Yaskawa INFORM job: Hexagon_ROBODK.jbi

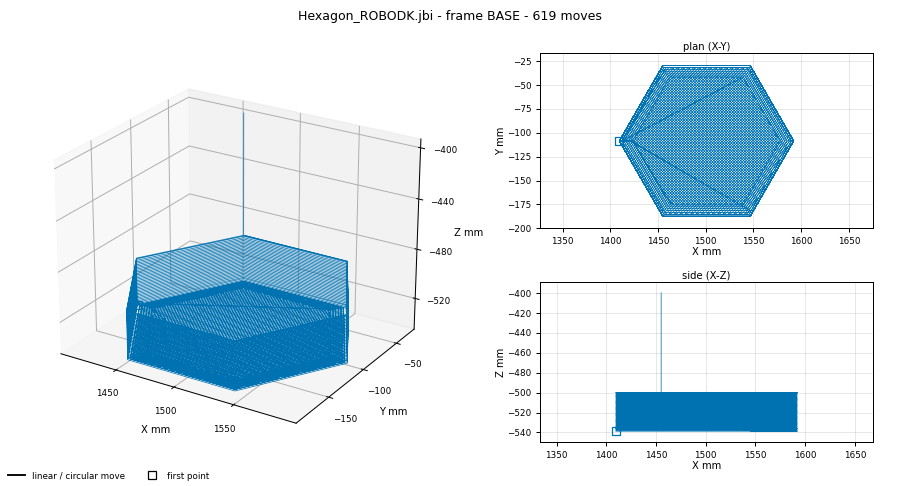
[picture p0: tool path of Hexagon_ROBODK.jbi in frame BASE, 619 of 620 moves have a stored position in this frame; points joined in program order, loops and branches not executed]
/JOB
//NAME HEXAGON
//POS
///NPOS 620,0,0,0,0,0
///TOOL 9
///POSTYPE PULSE
///PULSE
C00000=-4,42,-30,0,-18,-176
///TOOL 9
///POSTYPE BASE
///RECTAN
///RCONF 0,0,0,0,0,0,0,0
C00001=1409.577,-108.483,-538.800,180.00,-0.00,180.00
C00002=1455.188,-29.484,-538.800,180.00,-0.00,-180.00
C00003=1546.406,-29.484,-538.800,180.00,-0.00,-180.00
C00004=1592.017,-108.483,-538.800,180.00,-0.00,180.00
C00005=1546.406,-187.483,-538.800,180.00,0.00,-180.00
C00006=1455.188,-187.483,-538.800,180.00,0.00,-180.00
C00007=1409.577,-108.483,-538.800,180.00,-0.00,180.00
C00008=1410.014,-107.726,-538.800,180.00,0.00,-180.00
C00009=1412.706,-108.484,-538.800,180.00,-0.00,-180.00
C00010=1411.773,-108.482,-538.800,180.00,-0.00,-180.00
C00011=1456.286,-31.385,-538.800,180.00,0.00,-180.00
C00012=1545.308,-31.385,-538.800,180.00,-0.00,-180.00
C00013=1589.821,-108.483,-538.800,180.00,0.00,180.00
C00014=1545.308,-185.582,-538.800,180.00,-0.00,-180.00
C00015=1456.286,-185.582,-538.800,180.00,-0.00,180.00
C00016=1411.773,-108.482,-538.800,180.00,-0.00,-180.00
C00017=1412.706,-108.484,-538.800,180.00,-0.00,-180.00
C00018=1458.101,-32.386,-538.800,180.00,0.00,-180.00
C00019=1455.169,-35.318,-538.800,180.00,0.00,-180.00
C00020=1454.816,-35.671,-538.800,180.00,0.00,180.00
C00021=1460.929,-32.386,-538.800,180.00,0.00,-180.00
C00022=1451.306,-42.010,-538.800,180.00,-0.00,-180.00
C00023=1450.953,-42.363,-538.800,180.00,-0.00,-180.00
C00024=1447.442,-48.702,-538.800,180.00,-0.00,-180.00
C00025=1463.758,-32.386,-538.800,180.00,0.00,180.00
C00026=1466.586,-32.386,-538.800,180.00,0.00,180.00
C00027=1443.578,-55.394,-538.800,180.00,0.00,-180.00
C00028=1443.225,-55.747,-538.800,180.00,0.00,-180.00
C00029=1439.715,-62.086,-538.800,180.00,-0.00,180.00
C00030=1469.415,-32.386,-538.800,180.00,-0.00,-180.00
C00031=1472.243,-32.386,-538.800,180.00,-0.00,-180.00
C00032=1435.850,-68.779,-538.800,180.00,-0.00,-180.00
C00033=1435.497,-69.132,-538.800,180.00,0.00,-180.00
C00034=1431.987,-75.471,-538.800,180.00,0.00,180.00
C00035=1475.071,-32.386,-538.800,180.00,-0.00,-180.00
C00036=1477.900,-32.386,-538.800,180.00,0.00,180.00
C00037=1428.123,-82.163,-538.800,180.00,0.00,180.00
C00038=1427.770,-82.516,-538.800,180.00,0.00,-180.00
C00039=1424.259,-88.855,-538.800,180.00,-0.00,180.00
C00040=1480.728,-32.386,-538.800,180.00,0.00,180.00
C00041=1483.557,-32.386,-538.800,180.00,-0.00,-180.00
C00042=1420.396,-95.547,-538.800,180.00,0.00,180.00
C00043=1420.043,-95.900,-538.800,180.00,-0.00,-180.00
C00044=1416.532,-102.239,-538.800,180.00,0.00,-180.00
C00045=1486.385,-32.386,-538.800,180.00,-0.00,180.00
C00046=1489.214,-32.386,-538.800,180.00,-0.00,180.00
C00047=1412.997,-108.603,-538.800,180.00,0.00,-180.00
C00048=1414.032,-110.396,-538.800,180.00,0.00,-180.00
C00049=1492.042,-32.386,-538.800,180.00,0.00,-180.00
C00050=1494.870,-32.386,-538.800,180.00,0.00,-180.00
C00051=1415.067,-112.190,-538.800,180.00,0.00,-180.00
C00052=1416.102,-113.983,-538.800,180.00,0.00,-180.00
C00053=1497.699,-32.386,-538.800,180.00,0.00,-180.00
C00054=1500.527,-32.386,-538.800,180.00,-0.00,-180.00
C00055=1417.137,-115.776,-538.800,180.00,-0.00,-180.00
C00056=1418.173,-117.569,-538.800,180.00,0.00,180.00
C00057=1503.356,-32.386,-538.800,180.00,0.00,-180.00
C00058=1506.184,-32.386,-538.800,180.00,-0.00,-180.00
C00059=1419.208,-119.362,-538.800,180.00,0.00,-180.00
C00060=1420.243,-121.156,-538.800,180.00,-0.00,-180.00
C00061=1509.013,-32.386,-538.800,180.00,-0.00,-180.00
C00062=1511.841,-32.386,-538.800,180.00,0.00,180.00
C00063=1421.278,-122.949,-538.800,180.00,0.00,-180.00
C00064=1422.313,-124.742,-538.800,180.00,-0.00,-180.00
C00065=1514.669,-32.386,-538.800,180.00,-0.00,-180.00
C00066=1517.498,-32.386,-538.800,180.00,0.00,-180.00
C00067=1423.349,-126.535,-538.800,180.00,-0.00,-180.00
C00068=1424.384,-128.329,-538.800,180.00,0.00,180.00
C00069=1520.326,-32.386,-538.800,180.00,-0.00,-180.00
C00070=1523.155,-32.386,-538.800,180.00,0.00,-180.00
C00071=1425.419,-130.122,-538.800,180.00,-0.00,180.00
C00072=1426.455,-131.914,-538.800,180.00,-0.00,-180.00
C00073=1525.983,-32.386,-538.800,180.00,0.00,-180.00
C00074=1528.812,-32.386,-538.800,180.00,-0.00,-180.00
C00075=1427.490,-133.708,-538.800,180.00,0.00,-180.00
C00076=1428.525,-135.501,-538.800,180.00,0.00,-180.00
C00077=1531.640,-32.386,-538.800,180.00,-0.00,180.00
C00078=1534.468,-32.386,-538.800,180.00,0.00,-180.00
C00079=1429.561,-137.294,-538.800,180.00,0.00,-180.00
C00080=1430.596,-139.087,-538.800,180.00,-0.00,180.00
C00081=1537.297,-32.386,-538.800,180.00,-0.00,-180.00
C00082=1540.125,-32.386,-538.800,180.00,0.00,-180.00
C00083=1431.631,-140.880,-538.800,180.00,0.00,180.00
C00084=1432.666,-142.674,-538.800,180.00,0.00,180.00
C00085=1542.954,-32.386,-538.800,180.00,-0.00,-180.00
C00086=1545.115,-33.053,-538.800,180.00,-0.00,-180.00
C00087=1433.701,-144.467,-538.800,180.00,-0.00,-180.00
C00088=1434.737,-146.260,-538.800,180.00,-0.00,-180.00
C00089=1546.150,-34.846,-538.800,180.00,0.00,-180.00
C00090=1547.186,-36.639,-538.800,180.00,0.00,180.00
C00091=1435.772,-148.053,-538.800,180.00,-0.00,-180.00
C00092=1436.807,-149.847,-538.800,180.00,0.00,-180.00
C00093=1548.221,-38.433,-538.800,180.00,-0.00,-180.00
C00094=1549.257,-40.225,-538.800,180.00,0.00,-180.00
C00095=1437.842,-151.640,-538.800,180.00,0.00,180.00
C00096=1438.877,-153.433,-538.800,180.00,-0.00,-180.00
C00097=1550.292,-42.018,-538.800,180.00,0.00,180.00
C00098=1551.327,-43.812,-538.800,180.00,0.00,-180.00
C00099=1439.913,-155.226,-538.800,180.00,0.00,-180.00
C00100=1440.949,-157.019,-538.800,180.00,0.00,180.00
C00101=1552.362,-45.605,-538.800,180.00,0.00,180.00
C00102=1553.398,-47.398,-538.800,180.00,-0.00,-180.00
C00103=1441.984,-158.812,-538.800,180.00,-0.00,-180.00
C00104=1443.019,-160.605,-538.800,180.00,0.00,-180.00
C00105=1554.433,-49.191,-538.800,180.00,0.00,-180.00
C00106=1555.468,-50.985,-538.800,180.00,0.00,-180.00
C00107=1444.054,-162.398,-538.800,180.00,-0.00,-180.00
C00108=1445.089,-164.192,-538.800,180.00,-0.00,180.00
C00109=1556.503,-52.778,-538.800,180.00,-0.00,180.00
C00110=1557.538,-54.571,-538.800,180.00,-0.00,-180.00
C00111=1446.125,-165.985,-538.800,180.00,0.00,-180.00
C00112=1447.160,-167.778,-538.800,180.00,0.00,-180.00
C00113=1558.574,-56.364,-538.800,180.00,0.00,-180.00
C00114=1559.610,-58.157,-538.800,180.00,-0.00,180.00
C00115=1448.195,-169.571,-538.800,180.00,-0.00,-180.00
C00116=1449.230,-171.365,-538.800,180.00,0.00,180.00
C00117=1560.645,-59.950,-538.800,180.00,0.00,-180.00
C00118=1561.680,-61.743,-538.800,180.00,0.00,-180.00
C00119=1450.265,-173.158,-538.800,180.00,0.00,180.00
C00120=1451.301,-174.951,-538.800,180.00,-0.00,-180.00
C00121=1562.715,-63.536,-538.800,180.00,0.00,180.00
C00122=1563.750,-65.330,-538.800,180.00,0.00,-180.00
C00123=1452.336,-176.744,-538.800,180.00,-0.00,-180.00
C00124=1453.371,-178.537,-538.800,180.00,-0.00,-180.00
C00125=1564.786,-67.123,-538.800,180.00,0.00,-180.00
C00126=1565.821,-68.916,-538.800,180.00,-0.00,-180.00
C00127=1454.406,-180.331,-538.800,180.00,0.00,-180.00
C00128=1455.442,-182.123,-538.800,180.00,-0.00,-180.00
C00129=1566.857,-70.709,-538.800,180.00,0.00,180.00
C00130=1567.892,-72.502,-538.800,180.00,-0.00,-180.00
C00131=1456.477,-183.916,-538.800,180.00,0.00,-180.00
C00132=1458.640,-184.582,-538.800,180.00,0.00,180.00
C00133=1568.927,-74.295,-538.800,180.00,0.00,-180.00
C00134=1569.962,-76.088,-538.800,180.00,0.00,-180.00
C00135=1461.468,-184.582,-538.800,180.00,-0.00,-180.00
C00136=1464.297,-184.582,-538.800,180.00,0.00,-180.00
C00137=1570.998,-77.881,-538.800,180.00,-0.00,180.00
C00138=1572.033,-79.675,-538.800,180.00,0.00,-180.00
C00139=1467.125,-184.582,-538.800,180.00,-0.00,-180.00
C00140=1469.953,-184.582,-538.800,180.00,0.00,180.00
C00141=1573.068,-81.468,-538.800,180.00,-0.00,-180.00
C00142=1574.103,-83.261,-538.800,180.00,-0.00,-180.00
C00143=1472.782,-184.582,-538.800,180.00,-0.00,180.00
C00144=1475.610,-184.582,-538.800,180.00,0.00,-180.00
C00145=1575.138,-85.054,-538.800,180.00,0.00,180.00
C00146=1576.174,-86.847,-538.800,180.00,0.00,-180.00
C00147=1478.439,-184.582,-538.800,180.00,0.00,-180.00
C00148=1481.267,-184.582,-538.800,180.00,0.00,-180.00
C00149=1577.209,-88.640,-538.800,180.00,-0.00,-180.00
C00150=1578.245,-90.433,-538.800,180.00,-0.00,-180.00
C00151=1484.095,-184.582,-538.800,180.00,0.00,-180.00
C00152=1486.924,-184.582,-538.800,180.00,-0.00,180.00
C00153=1579.280,-92.227,-538.800,180.00,0.00,-180.00
C00154=1580.315,-94.020,-538.800,180.00,0.00,-180.00
C00155=1489.752,-184.582,-538.800,180.00,0.00,-180.00
C00156=1492.581,-184.582,-538.800,180.00,-0.00,-180.00
C00157=1581.350,-95.813,-538.800,180.00,-0.00,-180.00
C00158=1582.385,-97.606,-538.800,180.00,0.00,180.00
C00159=1495.409,-184.582,-538.800,180.00,-0.00,-180.00
C00160=1498.238,-184.582,-538.800,180.00,0.00,180.00
C00161=1583.421,-99.399,-538.800,180.00,0.00,-180.00
C00162=1584.456,-101.193,-538.800,180.00,-0.00,-180.00
C00163=1501.066,-184.582,-538.800,180.00,0.00,-180.00
C00164=1503.894,-184.582,-538.800,180.00,-0.00,-180.00
C00165=1585.492,-102.985,-538.800,180.00,0.00,180.00
C00166=1586.527,-104.778,-538.800,180.00,0.00,-180.00
C00167=1506.723,-184.582,-538.800,180.00,-0.00,-180.00
C00168=1509.551,-184.582,-538.800,180.00,0.00,-180.00
C00169=1587.562,-106.572,-538.800,180.00,0.00,-180.00
C00170=1588.597,-108.365,-538.800,180.00,0.00,-180.00
C00171=1512.380,-184.582,-538.800,180.00,0.00,-180.00
C00172=1515.208,-184.582,-538.800,180.00,0.00,-180.00
C00173=1585.057,-114.734,-538.800,180.00,0.00,180.00
C00174=1585.410,-114.381,-538.800,180.00,0.00,-180.00
C00175=1581.193,-121.426,-538.800,180.00,-0.00,-180.00
C00176=1518.037,-184.582,-538.800,180.00,-0.00,-180.00
C00177=1520.865,-184.582,-538.800,180.00,-0.00,-180.00
C00178=1577.330,-128.118,-538.800,180.00,0.00,-180.00
C00179=1577.683,-127.765,-538.800,180.00,0.00,-180.00
C00180=1573.466,-134.810,-538.800,180.00,-0.00,-180.00
C00181=1523.693,-184.582,-538.800,180.00,-0.00,-180.00
C00182=1526.522,-184.582,-538.800,180.00,0.00,-180.00
C00183=1569.602,-141.502,-538.800,180.00,0.00,180.00
C00184=1569.955,-141.149,-538.800,180.00,0.00,180.00
C00185=1565.739,-148.194,-538.800,180.00,0.00,-180.00
C00186=1529.350,-184.582,-538.800,180.00,0.00,-180.00
C00187=1532.179,-184.582,-538.800,180.00,0.00,-180.00
C00188=1561.875,-154.886,-538.800,180.00,-0.00,-180.00
C00189=1562.228,-154.533,-538.800,180.00,0.00,180.00
C00190=1558.011,-161.578,-538.800,180.00,0.00,-180.00
C00191=1535.007,-184.582,-538.800,180.00,0.00,-180.00
C00192=1537.836,-184.582,-538.800,180.00,-0.00,180.00
C00193=1554.148,-168.270,-538.800,180.00,-0.00,-180.00
C00194=1554.501,-167.917,-538.800,180.00,-0.00,-180.00
C00195=1550.284,-174.962,-538.800,180.00,-0.00,-180.00
C00196=1540.664,-184.582,-538.800,180.00,-0.00,-180.00
C00197=1543.492,-184.582,-538.800,180.00,0.00,-180.00
C00198=1546.421,-181.654,-538.800,180.00,0.00,-180.00
C00199=1546.774,-181.301,-538.800,180.00,-0.00,180.00
C00200=1545.171,-180.377,-538.800,180.00,-0.00,-180.00
C00201=1545.171,-180.377,-537.600,180.00,0.00,-180.00
C00202=1421.124,-108.483,-537.600,180.00,0.00,180.00
C00203=1441.043,-73.984,-537.600,180.00,0.00,-180.00
C00204=1460.961,-39.484,-537.600,180.00,0.00,180.00
C00205=1540.633,-39.484,-537.600,180.00,0.00,-180.00
C00206=1580.470,-108.483,-537.600,180.00,0.00,-180.00
C00207=1540.633,-177.483,-537.600,180.00,-0.00,-180.00
C00208=1460.961,-177.483,-537.600,180.00,0.00,180.00
C00209=1421.124,-108.483,-537.600,180.00,0.00,180.00
C00210=1418.815,-108.483,-537.600,180.00,0.00,-180.00
C00211=1439.311,-72.984,-537.600,180.00,-0.00,-180.00
C00212=1459.807,-37.484,-537.600,180.00,0.00,-180.00
C00213=1541.787,-37.484,-537.600,180.00,0.00,-180.00
C00214=1582.779,-108.483,-537.600,180.00,0.00,180.00
C00215=1541.787,-179.483,-537.600,180.00,0.00,180.00
C00216=1459.807,-179.483,-537.600,180.00,0.00,-180.00
C00217=1418.815,-108.483,-537.600,180.00,0.00,-180.00
C00218=1416.506,-108.483,-537.600,180.00,-0.00,-180.00
C00219=1437.579,-71.984,-537.600,180.00,-0.00,-180.00
C00220=1458.652,-35.484,-537.600,180.00,0.00,180.00
C00221=1542.942,-35.484,-537.600,180.00,0.00,180.00
C00222=1585.088,-108.483,-537.600,180.00,-0.00,-180.00
C00223=1542.942,-181.483,-537.600,180.00,-0.00,-180.00
C00224=1458.652,-181.483,-537.600,180.00,0.00,-180.00
C00225=1416.506,-108.483,-537.600,180.00,-0.00,-180.00
C00226=1414.196,-108.483,-537.600,180.00,-0.00,180.00
C00227=1435.847,-70.984,-537.600,180.00,-0.00,-180.00
C00228=1457.497,-33.484,-537.600,180.00,0.00,-180.00
C00229=1544.097,-33.484,-537.600,180.00,0.00,-180.00
C00230=1587.398,-108.483,-537.600,180.00,0.00,180.00
C00231=1544.097,-183.483,-537.600,180.00,0.00,-180.00
C00232=1457.497,-183.483,-537.600,180.00,-0.00,-180.00
C00233=1414.196,-108.483,-537.600,180.00,-0.00,180.00
C00234=1412.706,-108.484,-537.600,180.00,0.00,-180.00
C00235=1411.887,-108.483,-537.600,180.00,-0.00,-180.00
C00236=1434.115,-69.984,-537.600,180.00,-0.00,180.00
C00237=1456.343,-31.484,-537.600,180.00,0.00,-180.00
C00238=1545.251,-31.484,-537.600,180.00,0.00,-180.00
C00239=1589.707,-108.483,-537.600,180.00,0.00,-180.00
C00240=1545.251,-185.483,-537.600,180.00,0.00,180.00
C00241=1456.343,-185.483,-537.600,180.00,0.00,-180.00
C00242=1411.887,-108.483,-537.600,180.00,-0.00,-180.00
C00243=1412.706,-108.484,-537.600,180.00,0.00,-180.00
C00244=1409.577,-108.483,-537.600,180.00,0.00,180.00
C00245=1432.383,-68.984,-537.600,180.00,-0.00,-180.00
C00246=1455.188,-29.484,-537.600,180.00,0.00,-180.00
C00247=1546.406,-29.484,-537.600,180.00,0.00,-180.00
C00248=1592.017,-108.483,-537.600,180.00,0.00,180.00
C00249=1546.406,-187.483,-537.600,180.00,0.00,-180.00
C00250=1455.188,-187.483,-537.600,180.00,0.00,-180.00
C00251=1409.577,-108.483,-537.600,180.00,0.00,180.00
C00252=1410.014,-107.726,-537.600,180.00,0.00,-180.00
C00253=1412.706,-108.484,-537.600,180.00,0.00,-180.00
C00254=1423.320,-108.483,-537.600,180.00,-0.00,180.00
C00255=1462.060,-41.384,-537.600,180.00,0.00,-180.00
C00256=1539.534,-41.384,-537.600,180.00,-0.00,-180.00
C00257=1578.274,-108.482,-537.600,180.00,0.00,180.00
C00258=1539.534,-175.582,-537.600,180.00,-0.00,-180.00
C00259=1462.060,-175.582,-537.600,180.00,0.00,-180.00
C00260=1423.320,-108.483,-537.600,180.00,-0.00,180.00
C00261=1463.506,-174.583,-537.600,180.00,0.00,-180.00
C00262=1461.448,-172.525,-537.600,180.00,0.00,-180.00
C00263=1466.334,-174.583,-537.600,180.00,-0.00,-180.00
C00264=1457.585,-165.833,-537.600,180.00,0.00,180.00
C00265=1457.232,-165.480,-537.600,180.00,0.00,-180.00
C00266=1453.721,-159.141,-537.600,180.00,-0.00,-180.00
C00267=1469.163,-174.583,-537.600,180.00,-0.00,-180.00
C00268=1471.991,-174.583,-537.600,180.00,0.00,180.00
C00269=1449.857,-152.449,-537.600,180.00,0.00,-180.00
C00270=1449.504,-152.096,-537.600,180.00,0.00,-180.00
C00271=1445.994,-145.757,-537.600,180.00,-0.00,-180.00
C00272=1474.820,-174.583,-537.600,180.00,0.00,180.00
C00273=1477.648,-174.583,-537.600,180.00,0.00,-180.00
C00274=1442.130,-139.065,-537.600,180.00,-0.00,-180.00
C00275=1441.777,-138.712,-537.600,180.00,-0.00,180.00
C00276=1438.266,-132.373,-537.600,180.00,0.00,-180.00
C00277=1480.477,-174.583,-537.600,180.00,0.00,-180.00
C00278=1483.305,-174.583,-537.600,180.00,-0.00,180.00
C00279=1434.403,-125.680,-537.600,180.00,-0.00,-180.00
C00280=1434.050,-125.327,-537.600,180.00,0.00,180.00
C00281=1430.539,-118.988,-537.600,180.00,0.00,180.00
C00282=1486.133,-174.583,-537.600,180.00,0.00,180.00
C00283=1488.962,-174.583,-537.600,180.00,-0.00,-180.00
C00284=1426.675,-112.296,-537.600,180.00,-0.00,-180.00
C00285=1426.322,-111.943,-537.600,180.00,0.00,-180.00
C00286=1424.921,-107.713,-537.600,180.00,0.00,-180.00
C00287=1491.790,-174.583,-537.600,180.00,0.00,-180.00
C00288=1494.619,-174.583,-537.600,180.00,0.00,-180.00
C00289=1425.956,-105.920,-537.600,180.00,-0.00,-180.00
C00290=1426.991,-104.126,-537.600,180.00,-0.00,-180.00
C00291=1497.447,-174.583,-537.600,180.00,-0.00,-180.00
C00292=1500.276,-174.583,-537.600,180.00,-0.00,-180.00
C00293=1428.026,-102.333,-537.600,180.00,-0.00,-180.00
C00294=1429.061,-100.540,-537.600,180.00,-0.00,180.00
C00295=1503.104,-174.583,-537.600,180.00,-0.00,-180.00
C00296=1505.932,-174.583,-537.600,180.00,-0.00,180.00
C00297=1430.097,-98.747,-537.600,180.00,0.00,-180.00
C00298=1431.132,-96.954,-537.600,180.00,-0.00,180.00
C00299=1508.761,-174.583,-537.600,180.00,0.00,-180.00
C00300=1511.589,-174.583,-537.600,180.00,-0.00,-180.00
C00301=1432.168,-95.161,-537.600,180.00,0.00,180.00
C00302=1433.203,-93.368,-537.600,180.00,-0.00,-180.00
C00303=1514.418,-174.583,-537.600,180.00,-0.00,180.00
C00304=1517.246,-174.583,-537.600,180.00,0.00,-180.00
C00305=1434.238,-91.575,-537.600,180.00,0.00,180.00
C00306=1435.273,-89.781,-537.600,180.00,-0.00,-180.00
C00307=1520.075,-174.583,-537.600,180.00,-0.00,-180.00
C00308=1522.903,-174.583,-537.600,180.00,-0.00,-180.00
C00309=1436.309,-87.988,-537.600,180.00,-0.00,-180.00
C00310=1437.344,-86.195,-537.600,180.00,-0.00,-180.00
C00311=1525.731,-174.583,-537.600,180.00,0.00,180.00
C00312=1528.560,-174.583,-537.600,180.00,-0.00,180.00
C00313=1438.379,-84.402,-537.600,180.00,-0.00,-180.00
C00314=1439.414,-82.608,-537.600,180.00,0.00,180.00
C00315=1531.388,-174.583,-537.600,180.00,0.00,-180.00
C00316=1534.217,-174.583,-537.600,180.00,-0.00,-180.00
C00317=1440.449,-80.815,-537.600,180.00,0.00,180.00
C00318=1441.485,-79.023,-537.600,180.00,0.00,-180.00
C00319=1537.045,-174.583,-537.600,180.00,0.00,-180.00
C00320=1539.292,-174.001,-537.600,180.00,-0.00,180.00
C00321=1442.520,-77.230,-537.600,180.00,0.00,-180.00
C00322=1443.556,-75.436,-537.600,180.00,-0.00,-180.00
C00323=1540.327,-172.207,-537.600,180.00,-0.00,-180.00
C00324=1541.362,-170.414,-537.600,180.00,0.00,180.00
C00325=1444.591,-73.643,-537.600,180.00,0.00,-180.00
C00326=1445.626,-71.850,-537.600,180.00,0.00,-180.00
C00327=1542.397,-168.621,-537.600,180.00,0.00,-180.00
C00328=1543.432,-166.828,-537.600,180.00,0.00,-180.00
C00329=1446.661,-70.057,-537.600,180.00,-0.00,180.00
C00330=1447.696,-68.263,-537.600,180.00,0.00,180.00
C00331=1544.468,-165.035,-537.600,180.00,0.00,180.00
C00332=1545.503,-163.241,-537.600,180.00,0.00,-180.00
C00333=1448.732,-66.470,-537.600,180.00,-0.00,-180.00
C00334=1449.767,-64.677,-537.600,180.00,0.00,180.00
C00335=1546.538,-161.448,-537.600,180.00,-0.00,-180.00
C00336=1547.573,-159.655,-537.600,180.00,-0.00,-180.00
C00337=1450.803,-62.884,-537.600,180.00,-0.00,-180.00
C00338=1451.838,-61.091,-537.600,180.00,0.00,180.00
C00339=1548.608,-157.862,-537.600,180.00,-0.00,-180.00
C00340=1549.644,-156.068,-537.600,180.00,-0.00,-180.00
C00341=1452.873,-59.298,-537.600,180.00,-0.00,180.00
C00342=1453.908,-57.505,-537.600,180.00,0.00,180.00
C00343=1550.679,-154.275,-537.600,180.00,-0.00,-180.00
C00344=1551.715,-152.483,-537.600,180.00,0.00,-180.00
C00345=1454.944,-55.712,-537.600,180.00,-0.00,-180.00
C00346=1455.979,-53.918,-537.600,180.00,0.00,-180.00
C00347=1552.750,-150.689,-537.600,180.00,0.00,-180.00
C00348=1553.785,-148.896,-537.600,180.00,-0.00,-180.00
C00349=1457.014,-52.125,-537.600,180.00,0.00,-180.00
C00350=1458.049,-50.332,-537.600,180.00,-0.00,-180.00
C00351=1554.820,-147.103,-537.600,180.00,-0.00,-180.00
C00352=1555.856,-145.310,-537.600,180.00,0.00,-180.00
C00353=1459.084,-48.539,-537.600,180.00,0.00,-180.00
C00354=1460.120,-46.746,-537.600,180.00,-0.00,-180.00
C00355=1556.891,-143.517,-537.600,180.00,0.00,180.00
C00356=1557.926,-141.723,-537.600,180.00,0.00,-180.00
C00357=1461.156,-44.953,-537.600,180.00,-0.00,-180.00
C00358=1462.191,-43.160,-537.600,180.00,-0.00,-180.00
C00359=1558.961,-139.930,-537.600,180.00,0.00,180.00
C00360=1559.996,-138.137,-537.600,180.00,-0.00,180.00
C00361=1464.245,-42.385,-537.600,180.00,0.00,180.00
C00362=1467.073,-42.385,-537.600,180.00,0.00,-180.00
C00363=1561.032,-136.344,-537.600,180.00,-0.00,-180.00
C00364=1562.067,-134.550,-537.600,180.00,-0.00,-180.00
C00365=1469.902,-42.385,-537.600,180.00,-0.00,-180.00
C00366=1472.730,-42.385,-537.600,180.00,0.00,-180.00
C00367=1563.102,-132.757,-537.600,180.00,-0.00,180.00
C00368=1564.138,-130.965,-537.600,180.00,-0.00,180.00
C00369=1475.559,-42.385,-537.600,180.00,0.00,-180.00
C00370=1478.387,-42.385,-537.600,180.00,0.00,-180.00
C00371=1565.173,-129.171,-537.600,180.00,-0.00,180.00
C00372=1566.208,-127.378,-537.600,180.00,0.00,-180.00
C00373=1481.215,-42.385,-537.600,180.00,0.00,-180.00
C00374=1484.044,-42.385,-537.600,180.00,0.00,-180.00
C00375=1567.243,-125.585,-537.600,180.00,0.00,180.00
C00376=1568.279,-123.792,-537.600,180.00,0.00,-180.00
C00377=1486.872,-42.385,-537.600,180.00,0.00,-180.00
C00378=1489.701,-42.385,-537.600,180.00,0.00,180.00
C00379=1569.314,-121.999,-537.600,180.00,0.00,-180.00
C00380=1570.349,-120.205,-537.600,180.00,0.00,-180.00
C00381=1492.529,-42.385,-537.600,180.00,0.00,-180.00
C00382=1495.358,-42.385,-537.600,180.00,0.00,-180.00
C00383=1571.384,-118.412,-537.600,180.00,-0.00,-180.00
C00384=1572.420,-116.619,-537.600,180.00,0.00,180.00
C00385=1498.186,-42.385,-537.600,180.00,0.00,-180.00
C00386=1501.014,-42.385,-537.600,180.00,0.00,-180.00
C00387=1573.455,-114.826,-537.600,180.00,-0.00,-180.00
C00388=1574.490,-113.032,-537.600,180.00,0.00,180.00
C00389=1503.843,-42.385,-537.600,180.00,-0.00,-180.00
C00390=1506.671,-42.385,-537.600,180.00,0.00,-180.00
C00391=1575.525,-111.239,-537.600,180.00,0.00,-180.00
C00392=1576.561,-109.447,-537.600,180.00,0.00,180.00
C00393=1509.500,-42.385,-537.600,180.00,0.00,-180.00
C00394=1512.328,-42.385,-537.600,180.00,-0.00,-180.00
C00395=1575.330,-105.387,-537.600,180.00,-0.00,-180.00
C00396=1575.683,-105.740,-537.600,180.00,0.00,-180.00
C00397=1571.466,-98.695,-537.600,180.00,0.00,-180.00
C00398=1515.157,-42.385,-537.600,180.00,0.00,-180.00
C00399=1517.985,-42.385,-537.600,180.00,-0.00,-180.00
C00400=1567.603,-92.003,-537.600,180.00,0.00,-180.00
C00401=1567.956,-92.356,-537.600,180.00,0.00,-180.00
C00402=1563.739,-85.311,-537.600,180.00,0.00,-180.00
C00403=1520.813,-42.385,-537.600,180.00,-0.00,-180.00
C00404=1523.642,-42.385,-537.600,180.00,-0.00,180.00
C00405=1559.875,-78.619,-537.600,180.00,-0.00,180.00
C00406=1560.228,-78.972,-537.600,180.00,-0.00,180.00
C00407=1556.012,-71.927,-537.600,180.00,0.00,180.00
C00408=1526.470,-42.385,-537.600,180.00,0.00,-180.00
C00409=1529.299,-42.385,-537.600,180.00,-0.00,180.00
C00410=1552.148,-65.235,-537.600,180.00,0.00,-180.00
C00411=1552.501,-65.588,-537.600,180.00,-0.00,180.00
C00412=1548.285,-58.543,-537.600,180.00,0.00,-180.00
C00413=1532.127,-42.385,-537.600,180.00,-0.00,180.00
C00414=1534.956,-42.385,-537.600,180.00,-0.00,180.00
C00415=1544.421,-51.851,-537.600,180.00,0.00,-180.00
C00416=1544.774,-52.204,-537.600,180.00,0.00,180.00
C00417=1540.557,-45.159,-537.600,180.00,0.00,180.00
C00418=1537.784,-42.385,-537.600,180.00,-0.00,180.00
C00419=1537.784,-42.385,-536.400,180.00,0.00,180.00
C00420=1412.706,-108.484,-536.400,180.00,-0.00,-180.00
C00421=1409.576,-108.484,-536.400,180.00,-0.00,-180.00
C00422=1455.186,-187.484,-536.400,180.00,-0.00,-180.00
C00423=1546.408,-187.484,-536.400,180.00,0.00,180.00
C00424=1592.018,-108.484,-536.400,180.00,0.00,180.00
C00425=1546.408,-29.484,-536.400,180.00,0.00,-180.00
C00426=1455.186,-29.484,-536.400,180.00,-0.00,-180.00
C00427=1409.576,-108.484,-536.400,180.00,-0.00,-180.00
C00428=1455.186,-187.484,-536.200,180.00,0.00,-180.00
C00429=1546.408,-187.484,-536.000,180.00,0.00,180.00
C00430=1592.018,-108.484,-535.800,180.00,-0.00,180.00
C00431=1546.408,-29.484,-535.600,180.00,0.00,-180.00
C00432=1455.186,-29.484,-535.400,180.00,-0.00,-180.00
C00433=1409.576,-108.484,-535.200,180.00,-0.00,-180.00
C00434=1455.186,-187.484,-535.000,180.00,0.00,-180.00
C00435=1546.408,-187.484,-534.800,180.00,-0.00,-180.00
C00436=1592.018,-108.484,-534.600,180.00,-0.00,180.00
C00437=1546.408,-29.484,-534.400,180.00,-0.00,-180.00
C00438=1455.186,-29.484,-534.200,180.00,0.00,-180.00
C00439=1409.576,-108.484,-534.000,180.00,0.00,-180.00
C00440=1455.186,-187.484,-533.800,180.00,0.00,-180.00
C00441=1546.408,-187.484,-533.600,180.00,0.00,-180.00
C00442=1592.018,-108.484,-533.400,180.00,0.00,180.00
C00443=1546.408,-29.484,-533.200,180.00,-0.00,-180.00
C00444=1455.186,-29.484,-533.000,180.00,-0.00,-180.00
C00445=1409.576,-108.484,-532.800,180.00,0.00,-180.00
C00446=1455.186,-187.484,-532.600,180.00,0.00,-180.00
C00447=1546.408,-187.484,-532.400,180.00,0.00,-180.00
C00448=1592.018,-108.484,-532.200,180.00,-0.00,180.00
C00449=1546.408,-29.484,-532.000,180.00,0.00,-180.00
C00450=1455.186,-29.484,-531.800,180.00,0.00,-180.00
C00451=1409.576,-108.484,-531.600,180.00,-0.00,-180.00
C00452=1455.186,-187.484,-531.400,180.00,-0.00,-180.00
C00453=1546.408,-187.484,-531.200,180.00,0.00,-180.00
C00454=1592.018,-108.484,-531.000,180.00,-0.00,180.00
C00455=1546.408,-29.484,-530.800,180.00,0.00,-180.00
C00456=1455.186,-29.484,-530.600,180.00,0.00,-180.00
C00457=1409.576,-108.484,-530.400,180.00,0.00,-180.00
C00458=1455.186,-187.484,-530.200,180.00,0.00,-180.00
C00459=1546.408,-187.484,-530.000,180.00,0.00,180.00
C00460=1592.018,-108.484,-529.800,180.00,0.00,180.00
C00461=1546.408,-29.484,-529.600,180.00,0.00,-180.00
C00462=1455.186,-29.484,-529.400,180.00,-0.00,-180.00
C00463=1409.576,-108.484,-529.200,180.00,-0.00,-180.00
C00464=1455.186,-187.484,-529.000,180.00,-0.00,-180.00
C00465=1546.408,-187.484,-528.800,180.00,-0.00,180.00
C00466=1592.018,-108.484,-528.600,180.00,0.00,180.00
C00467=1546.408,-29.484,-528.400,180.00,0.00,-180.00
C00468=1455.186,-29.484,-528.200,180.00,0.00,-180.00
C00469=1409.576,-108.484,-528.000,180.00,-0.00,-180.00
C00470=1455.186,-187.484,-527.800,180.00,-0.00,-180.00
C00471=1546.408,-187.484,-527.600,180.00,-0.00,-180.00
C00472=1592.018,-108.484,-527.400,180.00,-0.00,180.00
C00473=1546.408,-29.484,-527.200,180.00,0.00,-180.00
C00474=1455.186,-29.484,-527.000,180.00,0.00,-180.00
C00475=1409.576,-108.484,-526.800,180.00,0.00,-180.00
C00476=1455.186,-187.484,-526.600,180.00,0.00,-180.00
C00477=1546.408,-187.484,-526.400,180.00,-0.00,-180.00
C00478=1592.018,-108.484,-526.200,180.00,-0.00,180.00
C00479=1546.408,-29.484,-526.000,180.00,-0.00,-180.00
C00480=1455.186,-29.484,-525.800,180.00,0.00,-180.00
C00481=1409.576,-108.484,-525.600,180.00,0.00,-180.00
C00482=1455.186,-187.484,-525.400,180.00,0.00,-180.00
C00483=1546.408,-187.484,-525.200,180.00,-0.00,-180.00
C00484=1592.018,-108.484,-525.000,180.00,0.00,180.00
C00485=1546.408,-29.484,-524.800,180.00,-0.00,-180.00
C00486=1455.186,-29.484,-524.600,180.00,-0.00,-180.00
C00487=1409.576,-108.484,-524.400,180.00,0.00,-180.00
C00488=1455.186,-187.484,-524.200,180.00,0.00,-180.00
C00489=1546.408,-187.484,-524.000,180.00,0.00,-180.00
C00490=1592.018,-108.484,-523.800,180.00,-0.00,180.00
C00491=1546.408,-29.484,-523.600,180.00,0.00,-180.00
C00492=1455.186,-29.484,-523.400,180.00,0.00,-180.00
C00493=1409.576,-108.484,-523.200,180.00,-0.00,-180.00
C00494=1455.186,-187.484,-523.000,180.00,-0.00,-180.00
C00495=1546.408,-187.484,-522.800,180.00,0.00,180.00
C00496=1592.018,-108.484,-522.600,180.00,-0.00,180.00
C00497=1546.408,-29.484,-522.400,180.00,-0.00,-180.00
C00498=1455.186,-29.484,-522.200,180.00,0.00,-180.00
C00499=1409.576,-108.484,-522.000,180.00,0.00,-180.00
C00500=1455.186,-187.484,-521.800,180.00,-0.00,-180.00
C00501=1546.408,-187.484,-521.600,180.00,0.00,-180.00
C00502=1592.018,-108.484,-521.400,180.00,0.00,180.00
C00503=1546.408,-29.484,-521.200,180.00,0.00,-180.00
C00504=1455.186,-29.484,-521.000,180.00,0.00,-180.00
C00505=1409.576,-108.484,-520.800,180.00,-0.00,-180.00
C00506=1455.186,-187.484,-520.600,180.00,-0.00,-180.00
C00507=1546.408,-187.484,-520.400,180.00,-0.00,-180.00
C00508=1592.018,-108.484,-520.200,180.00,0.00,180.00
C00509=1546.408,-29.484,-520.000,180.00,-0.00,-180.00
C00510=1455.186,-29.484,-519.800,180.00,-0.00,-180.00
C00511=1409.576,-108.484,-519.600,180.00,0.00,-180.00
C00512=1455.186,-187.484,-519.400,180.00,0.00,-180.00
C00513=1546.408,-187.484,-519.200,180.00,0.00,-180.00
C00514=1592.018,-108.484,-519.000,180.00,-0.00,180.00
C00515=1546.408,-29.484,-518.800,180.00,0.00,-180.00
C00516=1455.186,-29.484,-518.600,180.00,-0.00,-180.00
C00517=1409.576,-108.484,-518.400,180.00,-0.00,-180.00
C00518=1455.186,-187.484,-518.200,180.00,-0.00,-180.00
C00519=1546.408,-187.484,-518.000,180.00,-0.00,-180.00
C00520=1592.018,-108.484,-517.800,180.00,-0.00,180.00
C00521=1546.408,-29.484,-517.600,180.00,-0.00,-180.00
C00522=1455.186,-29.484,-517.400,180.00,-0.00,-180.00
C00523=1409.576,-108.484,-517.200,180.00,-0.00,-180.00
C00524=1455.186,-187.484,-517.000,180.00,0.00,-180.00
C00525=1546.408,-187.484,-516.800,180.00,-0.00,-180.00
C00526=1592.018,-108.484,-516.600,180.00,0.00,180.00
C00527=1546.408,-29.484,-516.400,180.00,0.00,-180.00
C00528=1455.186,-29.484,-516.200,180.00,-0.00,-180.00
C00529=1409.576,-108.484,-516.000,180.00,0.00,-180.00
C00530=1455.186,-187.484,-515.800,180.00,-0.00,-180.00
C00531=1546.408,-187.484,-515.600,180.00,-0.00,-180.00
C00532=1592.018,-108.484,-515.400,180.00,-0.00,180.00
C00533=1546.408,-29.484,-515.200,180.00,0.00,-180.00
C00534=1455.186,-29.484,-515.000,180.00,0.00,-180.00
C00535=1409.576,-108.484,-514.800,180.00,0.00,-180.00
C00536=1455.186,-187.484,-514.600,180.00,-0.00,-180.00
C00537=1546.408,-187.484,-514.400,180.00,0.00,-180.00
C00538=1592.018,-108.484,-514.200,180.00,-0.00,180.00
C00539=1546.408,-29.484,-514.000,180.00,0.00,-180.00
C00540=1455.186,-29.484,-513.800,180.00,-0.00,-180.00
C00541=1409.576,-108.484,-513.600,180.00,-0.00,-180.00
C00542=1455.186,-187.484,-513.400,180.00,0.00,-180.00
C00543=1546.408,-187.484,-513.200,180.00,-0.00,180.00
C00544=1592.018,-108.484,-513.000,180.00,-0.00,180.00
C00545=1546.408,-29.484,-512.800,180.00,0.00,-180.00
C00546=1455.186,-29.484,-512.600,180.00,0.00,-180.00
C00547=1409.576,-108.484,-512.400,180.00,0.00,-180.00
C00548=1455.186,-187.484,-512.200,180.00,0.00,-180.00
C00549=1546.408,-187.484,-512.000,180.00,-0.00,-180.00
C00550=1592.018,-108.484,-511.800,180.00,0.00,180.00
C00551=1546.408,-29.484,-511.600,180.00,0.00,-180.00
C00552=1455.186,-29.484,-511.400,180.00,0.00,-180.00
C00553=1409.576,-108.484,-511.200,180.00,0.00,-180.00
C00554=1455.186,-187.484,-511.000,180.00,0.00,-180.00
C00555=1546.408,-187.484,-510.800,180.00,0.00,180.00
C00556=1592.018,-108.484,-510.600,180.00,0.00,180.00
C00557=1546.408,-29.484,-510.400,180.00,-0.00,-180.00
C00558=1455.186,-29.484,-510.200,180.00,0.00,-180.00
C00559=1409.576,-108.484,-510.000,180.00,0.00,-180.00
C00560=1455.186,-187.484,-509.800,180.00,-0.00,-180.00
C00561=1546.408,-187.484,-509.600,180.00,-0.00,-180.00
C00562=1592.018,-108.484,-509.400,180.00,-0.00,180.00
C00563=1546.408,-29.484,-509.200,180.00,0.00,-180.00
C00564=1455.186,-29.484,-509.000,180.00,0.00,-180.00
C00565=1409.576,-108.484,-508.800,180.00,0.00,-180.00
C00566=1455.186,-187.484,-508.600,180.00,0.00,-180.00
C00567=1546.408,-187.484,-508.400,180.00,0.00,180.00
C00568=1592.018,-108.484,-508.200,180.00,0.00,180.00
C00569=1546.408,-29.484,-508.000,180.00,0.00,-180.00
C00570=1455.186,-29.484,-507.800,180.00,0.00,-180.00
C00571=1409.576,-108.484,-507.600,180.00,-0.00,-180.00
C00572=1455.186,-187.484,-507.400,180.00,0.00,-180.00
C00573=1546.408,-187.484,-507.200,180.00,0.00,-180.00
C00574=1592.018,-108.484,-507.000,180.00,-0.00,180.00
C00575=1546.408,-29.484,-506.800,180.00,0.00,-180.00
C00576=1455.186,-29.484,-506.600,180.00,-0.00,-180.00
C00577=1409.576,-108.484,-506.400,180.00,0.00,-180.00
C00578=1455.186,-187.484,-506.200,180.00,0.00,-180.00
C00579=1546.408,-187.484,-506.000,180.00,-0.00,-180.00
C00580=1592.018,-108.484,-505.800,180.00,-0.00,180.00
C00581=1546.408,-29.484,-505.600,180.00,-0.00,-180.00
C00582=1455.186,-29.484,-505.400,180.00,-0.00,-180.00
C00583=1409.576,-108.484,-505.200,180.00,-0.00,-180.00
C00584=1455.186,-187.484,-505.000,180.00,-0.00,-180.00
C00585=1546.408,-187.484,-504.800,180.00,0.00,-180.00
C00586=1592.018,-108.484,-504.600,180.00,0.00,180.00
C00587=1546.408,-29.484,-504.400,180.00,0.00,-180.00
C00588=1455.186,-29.484,-504.200,180.00,0.00,-180.00
C00589=1409.576,-108.484,-504.000,180.00,-0.00,-180.00
C00590=1455.186,-187.484,-503.800,180.00,-0.00,-180.00
C00591=1546.408,-187.484,-503.600,180.00,0.00,-180.00
C00592=1592.018,-108.484,-503.400,180.00,0.00,180.00
C00593=1546.408,-29.484,-503.200,180.00,0.00,-180.00
C00594=1455.186,-29.484,-503.000,180.00,-0.00,-180.00
C00595=1409.576,-108.484,-502.800,180.00,-0.00,-180.00
C00596=1455.186,-187.484,-502.600,180.00,0.00,-180.00
C00597=1546.408,-187.484,-502.400,180.00,-0.00,-180.00
C00598=1592.018,-108.484,-502.200,180.00,0.00,180.00
C00599=1546.408,-29.484,-502.000,180.00,0.00,-180.00
C00600=1455.186,-29.484,-501.800,180.00,0.00,-180.00
C00601=1409.576,-108.484,-501.600,180.00,-0.00,-180.00
C00602=1455.186,-187.484,-501.400,180.00,-0.00,-180.00
C00603=1546.408,-187.484,-501.200,180.00,0.00,-180.00
C00604=1592.018,-108.484,-501.000,180.00,0.00,180.00
C00605=1546.408,-29.484,-500.800,180.00,-0.00,-180.00
C00606=1455.186,-29.484,-500.600,180.00,-0.00,-180.00
C00607=1409.576,-108.484,-500.400,180.00,0.00,-180.00
C00608=1455.186,-187.484,-500.291,180.00,0.00,-180.00
C00609=1546.408,-187.484,-500.182,180.00,0.00,-180.00
C00610=1592.018,-108.484,-500.073,180.00,0.00,180.00
C00611=1546.408,-29.484,-499.964,180.00,-0.00,-180.00
C00612=1455.186,-29.484,-499.855,180.00,0.00,-180.00
C00613=1409.576,-108.484,-499.745,180.00,0.00,-180.00
C00614=1455.186,-187.484,-499.745,180.00,-0.00,-180.00
C00615=1546.408,-187.484,-499.745,180.00,0.00,-180.00
C00616=1592.018,-108.484,-499.745,180.00,0.00,180.00
C00617=1546.408,-29.484,-499.745,180.00,-0.00,-180.00
C00618=1455.186,-29.484,-499.745,180.00,0.00,-180.00
C00619=1455.186,-29.484,-399.745,180.00,0.00,-180.00
//INST
///DATE 2024/04/09 21:14
///ATTR SC,RW
///GROUP1 RB1
NOP
'Program generated by RoboDK v
'5.6.7 for Yaskawa GP88 on 09/
'04/2024 21:14:32
'Using nominal kinematics.
'Using base frame
'Using TOOL 9:
'0.000,0.000,0.000,0.00,0.00,0
'.00
MOVJ C00000 VJ=100.0
MOVL C00001 V=150.0
MOVL C00002 V=150.0
MOVL C00003 V=150.0
MOVL C00004 V=150.0
MOVL C00005 V=150.0
MOVL C00006 V=150.0
MOVL C00007 V=150.0
MOVL C00008 V=150.0
MOVL C00009 V=150.0
MOVL C00010 V=150.0
MOVL C00011 V=150.0
MOVL C00012 V=150.0
MOVL C00013 V=150.0
MOVL C00014 V=150.0
MOVL C00015 V=150.0
MOVL C00016 V=150.0
MOVL C00017 V=150.0
MOVL C00018 V=150.0
MOVL C00019 V=150.0
MOVL C00020 V=150.0
MOVL C00021 V=150.0
MOVL C00022 V=150.0
MOVL C00023 V=150.0
MOVL C00024 V=150.0
MOVL C00025 V=150.0
MOVL C00026 V=150.0
MOVL C00027 V=150.0
MOVL C00028 V=150.0
MOVL C00029 V=150.0
MOVL C00030 V=150.0
MOVL C00031 V=150.0
MOVL C00032 V=150.0
MOVL C00033 V=150.0
MOVL C00034 V=150.0
MOVL C00035 V=150.0
MOVL C00036 V=150.0
MOVL C00037 V=150.0
MOVL C00038 V=150.0
MOVL C00039 V=150.0
MOVL C00040 V=150.0
MOVL C00041 V=150.0
MOVL C00042 V=150.0
MOVL C00043 V=150.0
MOVL C00044 V=150.0
MOVL C00045 V=150.0
MOVL C00046 V=150.0
MOVL C00047 V=150.0
MOVL C00048 V=150.0
MOVL C00049 V=150.0
MOVL C00050 V=150.0
MOVL C00051 V=150.0
MOVL C00052 V=150.0
MOVL C00053 V=150.0
MOVL C00054 V=150.0
MOVL C00055 V=150.0
MOVL C00056 V=150.0
MOVL C00057 V=150.0
MOVL C00058 V=150.0
MOVL C00059 V=150.0
MOVL C00060 V=150.0
MOVL C00061 V=150.0
MOVL C00062 V=150.0
MOVL C00063 V=150.0
MOVL C00064 V=150.0
MOVL C00065 V=150.0
MOVL C00066 V=150.0
MOVL C00067 V=150.0
MOVL C00068 V=150.0
MOVL C00069 V=150.0
MOVL C00070 V=150.0
MOVL C00071 V=150.0
MOVL C00072 V=150.0
MOVL C00073 V=150.0
MOVL C00074 V=150.0
MOVL C00075 V=150.0
MOVL C00076 V=150.0
MOVL C00077 V=150.0
MOVL C00078 V=150.0
MOVL C00079 V=150.0
MOVL C00080 V=150.0
MOVL C00081 V=150.0
MOVL C00082 V=150.0
MOVL C00083 V=150.0
MOVL C00084 V=150.0
MOVL C00085 V=150.0
MOVL C00086 V=150.0
MOVL C00087 V=150.0
MOVL C00088 V=150.0
MOVL C00089 V=150.0
MOVL C00090 V=150.0
MOVL C00091 V=150.0
MOVL C00092 V=150.0
MOVL C00093 V=150.0
MOVL C00094 V=150.0
MOVL C00095 V=150.0
MOVL C00096 V=150.0
MOVL C00097 V=150.0
MOVL C00098 V=150.0
MOVL C00099 V=150.0
MOVL C00100 V=150.0
MOVL C00101 V=150.0
MOVL C00102 V=150.0
MOVL C00103 V=150.0
MOVL C00104 V=150.0
MOVL C00105 V=150.0
MOVL C00106 V=150.0
MOVL C00107 V=150.0
MOVL C00108 V=150.0
MOVL C00109 V=150.0
MOVL C00110 V=150.0
MOVL C00111 V=150.0
MOVL C00112 V=150.0
MOVL C00113 V=150.0
MOVL C00114 V=150.0
MOVL C00115 V=150.0
MOVL C00116 V=150.0
MOVL C00117 V=150.0
MOVL C00118 V=150.0
MOVL C00119 V=150.0
MOVL C00120 V=150.0
MOVL C00121 V=150.0
MOVL C00122 V=150.0
MOVL C00123 V=150.0
MOVL C00124 V=150.0
MOVL C00125 V=150.0
MOVL C00126 V=150.0
MOVL C00127 V=150.0
MOVL C00128 V=150.0
MOVL C00129 V=150.0
MOVL C00130 V=150.0
MOVL C00131 V=150.0
MOVL C00132 V=150.0
MOVL C00133 V=150.0
MOVL C00134 V=150.0
MOVL C00135 V=150.0
MOVL C00136 V=150.0
MOVL C00137 V=150.0
MOVL C00138 V=150.0
MOVL C00139 V=150.0
MOVL C00140 V=150.0
MOVL C00141 V=150.0
MOVL C00142 V=150.0
MOVL C00143 V=150.0
MOVL C00144 V=150.0
MOVL C00145 V=150.0
MOVL C00146 V=150.0
MOVL C00147 V=150.0
MOVL C00148 V=150.0
MOVL C00149 V=150.0
MOVL C00150 V=150.0
MOVL C00151 V=150.0
MOVL C00152 V=150.0
MOVL C00153 V=150.0
MOVL C00154 V=150.0
MOVL C00155 V=150.0
MOVL C00156 V=150.0
MOVL C00157 V=150.0
MOVL C00158 V=150.0
MOVL C00159 V=150.0
MOVL C00160 V=150.0
MOVL C00161 V=150.0
MOVL C00162 V=150.0
MOVL C00163 V=150.0
MOVL C00164 V=150.0
MOVL C00165 V=150.0
MOVL C00166 V=150.0
MOVL C00167 V=150.0
MOVL C00168 V=150.0
MOVL C00169 V=150.0
MOVL C00170 V=150.0
MOVL C00171 V=150.0
MOVL C00172 V=150.0
MOVL C00173 V=150.0
MOVL C00174 V=150.0
MOVL C00175 V=150.0
MOVL C00176 V=150.0
MOVL C00177 V=150.0
MOVL C00178 V=150.0
MOVL C00179 V=150.0
MOVL C00180 V=150.0
MOVL C00181 V=150.0
MOVL C00182 V=150.0
MOVL C00183 V=150.0
MOVL C00184 V=150.0
MOVL C00185 V=150.0
MOVL C00186 V=150.0
MOVL C00187 V=150.0
MOVL C00188 V=150.0
MOVL C00189 V=150.0
MOVL C00190 V=150.0
MOVL C00191 V=150.0
MOVL C00192 V=150.0
MOVL C00193 V=150.0
MOVL C00194 V=150.0
MOVL C00195 V=150.0
MOVL C00196 V=150.0
MOVL C00197 V=150.0
MOVL C00198 V=150.0
MOVL C00199 V=150.0
MOVL C00200 V=150.0
MOVL C00201 V=60.00
MOVL C00202 V=150.0
MOVL C00203 V=150.0
MOVL C00204 V=150.0
MOVL C00205 V=150.0
MOVL C00206 V=150.0
MOVL C00207 V=150.0
MOVL C00208 V=150.0
MOVL C00209 V=150.0
MOVL C00210 V=150.0
MOVL C00211 V=150.0
MOVL C00212 V=150.0
MOVL C00213 V=150.0
MOVL C00214 V=150.0
MOVL C00215 V=150.0
MOVL C00216 V=150.0
MOVL C00217 V=150.0
MOVL C00218 V=150.0
MOVL C00219 V=150.0
MOVL C00220 V=150.0
MOVL C00221 V=150.0
MOVL C00222 V=150.0
MOVL C00223 V=150.0
MOVL C00224 V=150.0
MOVL C00225 V=150.0
MOVL C00226 V=150.0
MOVL C00227 V=150.0
MOVL C00228 V=150.0
MOVL C00229 V=150.0
MOVL C00230 V=150.0
MOVL C00231 V=150.0
MOVL C00232 V=150.0
MOVL C00233 V=150.0
MOVL C00234 V=150.0
MOVL C00235 V=150.0
MOVL C00236 V=150.0
MOVL C00237 V=150.0
MOVL C00238 V=150.0
MOVL C00239 V=150.0
MOVL C00240 V=150.0
MOVL C00241 V=150.0
MOVL C00242 V=150.0
MOVL C00243 V=150.0
MOVL C00244 V=150.0
MOVL C00245 V=150.0
MOVL C00246 V=150.0
MOVL C00247 V=150.0
MOVL C00248 V=150.0
MOVL C00249 V=150.0
MOVL C00250 V=150.0
MOVL C00251 V=150.0
MOVL C00252 V=150.0
MOVL C00253 V=150.0
MOVL C00254 V=150.0
MOVL C00255 V=150.0
MOVL C00256 V=150.0
MOVL C00257 V=150.0
MOVL C00258 V=150.0
MOVL C00259 V=150.0
MOVL C00260 V=150.0
MOVL C00261 V=150.0
MOVL C00262 V=150.0
MOVL C00263 V=150.0
MOVL C00264 V=150.0
MOVL C00265 V=150.0
MOVL C00266 V=150.0
MOVL C00267 V=150.0
MOVL C00268 V=150.0
MOVL C00269 V=150.0
MOVL C00270 V=150.0
MOVL C00271 V=150.0
MOVL C00272 V=150.0
MOVL C00273 V=150.0
MOVL C00274 V=150.0
MOVL C00275 V=150.0
MOVL C00276 V=150.0
MOVL C00277 V=150.0
MOVL C00278 V=150.0
MOVL C00279 V=150.0
MOVL C00280 V=150.0
MOVL C00281 V=150.0
MOVL C00282 V=150.0
MOVL C00283 V=150.0
MOVL C00284 V=150.0
MOVL C00285 V=150.0
MOVL C00286 V=150.0
MOVL C00287 V=150.0
MOVL C00288 V=150.0
MOVL C00289 V=150.0
MOVL C00290 V=150.0
MOVL C00291 V=150.0
MOVL C00292 V=150.0
MOVL C00293 V=150.0
MOVL C00294 V=150.0
MOVL C00295 V=150.0
MOVL C00296 V=150.0
MOVL C00297 V=150.0
MOVL C00298 V=150.0
MOVL C00299 V=150.0
MOVL C00300 V=150.0
MOVL C00301 V=150.0
MOVL C00302 V=150.0
MOVL C00303 V=150.0
MOVL C00304 V=150.0
MOVL C00305 V=150.0
MOVL C00306 V=150.0
MOVL C00307 V=150.0
MOVL C00308 V=150.0
MOVL C00309 V=150.0
MOVL C00310 V=150.0
MOVL C00311 V=150.0
MOVL C00312 V=150.0
MOVL C00313 V=150.0
MOVL C00314 V=150.0
MOVL C00315 V=150.0
MOVL C00316 V=150.0
MOVL C00317 V=150.0
MOVL C00318 V=150.0
MOVL C00319 V=150.0
MOVL C00320 V=150.0
MOVL C00321 V=150.0
MOVL C00322 V=150.0
MOVL C00323 V=150.0
MOVL C00324 V=150.0
MOVL C00325 V=150.0
MOVL C00326 V=150.0
MOVL C00327 V=150.0
MOVL C00328 V=150.0
MOVL C00329 V=150.0
MOVL C00330 V=150.0
MOVL C00331 V=150.0
MOVL C00332 V=150.0
MOVL C00333 V=150.0
MOVL C00334 V=150.0
MOVL C00335 V=150.0
MOVL C00336 V=150.0
MOVL C00337 V=150.0
MOVL C00338 V=150.0
MOVL C00339 V=150.0
MOVL C00340 V=150.0
MOVL C00341 V=150.0
MOVL C00342 V=150.0
MOVL C00343 V=150.0
MOVL C00344 V=150.0
MOVL C00345 V=150.0
MOVL C00346 V=150.0
MOVL C00347 V=150.0
MOVL C00348 V=150.0
MOVL C00349 V=150.0
MOVL C00350 V=150.0
MOVL C00351 V=150.0
MOVL C00352 V=150.0
MOVL C00353 V=150.0
MOVL C00354 V=150.0
MOVL C00355 V=150.0
MOVL C00356 V=150.0
MOVL C00357 V=150.0
MOVL C00358 V=150.0
MOVL C00359 V=150.0
MOVL C00360 V=150.0
MOVL C00361 V=150.0
MOVL C00362 V=150.0
MOVL C00363 V=150.0
MOVL C00364 V=150.0
MOVL C00365 V=150.0
MOVL C00366 V=150.0
MOVL C00367 V=150.0
MOVL C00368 V=150.0
MOVL C00369 V=150.0
MOVL C00370 V=150.0
MOVL C00371 V=150.0
MOVL C00372 V=150.0
MOVL C00373 V=150.0
MOVL C00374 V=150.0
MOVL C00375 V=150.0
MOVL C00376 V=150.0
MOVL C00377 V=150.0
MOVL C00378 V=150.0
MOVL C00379 V=150.0
MOVL C00380 V=150.0
MOVL C00381 V=150.0
MOVL C00382 V=150.0
MOVL C00383 V=150.0
MOVL C00384 V=150.0
MOVL C00385 V=150.0
MOVL C00386 V=150.0
MOVL C00387 V=150.0
MOVL C00388 V=150.0
MOVL C00389 V=150.0
MOVL C00390 V=150.0
MOVL C00391 V=150.0
MOVL C00392 V=150.0
MOVL C00393 V=150.0
MOVL C00394 V=150.0
MOVL C00395 V=150.0
MOVL C00396 V=150.0
MOVL C00397 V=150.0
MOVL C00398 V=150.0
MOVL C00399 V=150.0
MOVL C00400 V=150.0
MOVL C00401 V=150.0
MOVL C00402 V=150.0
MOVL C00403 V=150.0
MOVL C00404 V=150.0
MOVL C00405 V=150.0
MOVL C00406 V=150.0
MOVL C00407 V=150.0
MOVL C00408 V=150.0
MOVL C00409 V=150.0
MOVL C00410 V=150.0
MOVL C00411 V=150.0
MOVL C00412 V=150.0
MOVL C00413 V=150.0
MOVL C00414 V=150.0
MOVL C00415 V=150.0
MOVL C00416 V=150.0
MOVL C00417 V=150.0
MOVL C00418 V=150.0
MOVL C00419 V=60.00
MOVL C00420 V=150.0
MOVL C00421 V=150.0
MOVL C00422 V=150.0
MOVL C00423 V=150.0
MOVL C00424 V=150.0
MOVL C00425 V=150.0
MOVL C00426 V=150.0
MOVL C00427 V=150.0
MOVL C00428 V=150.0
MOVL C00429 V=150.0
MOVL C00430 V=150.0
MOVL C00431 V=150.0
MOVL C00432 V=150.0
MOVL C00433 V=150.0
MOVL C00434 V=150.0
MOVL C00435 V=150.0
MOVL C00436 V=150.0
MOVL C00437 V=150.0
MOVL C00438 V=150.0
MOVL C00439 V=150.0
MOVL C00440 V=150.0
MOVL C00441 V=150.0
MOVL C00442 V=150.0
MOVL C00443 V=150.0
MOVL C00444 V=150.0
MOVL C00445 V=150.0
MOVL C00446 V=150.0
MOVL C00447 V=150.0
MOVL C00448 V=150.0
MOVL C00449 V=150.0
MOVL C00450 V=150.0
MOVL C00451 V=150.0
MOVL C00452 V=150.0
MOVL C00453 V=150.0
MOVL C00454 V=150.0
MOVL C00455 V=150.0
MOVL C00456 V=150.0
MOVL C00457 V=150.0
MOVL C00458 V=150.0
MOVL C00459 V=150.0
MOVL C00460 V=150.0
MOVL C00461 V=150.0
MOVL C00462 V=150.0
MOVL C00463 V=150.0
MOVL C00464 V=150.0
MOVL C00465 V=150.0
MOVL C00466 V=150.0
MOVL C00467 V=150.0
MOVL C00468 V=150.0
MOVL C00469 V=150.0
MOVL C00470 V=150.0
MOVL C00471 V=150.0
MOVL C00472 V=150.0
MOVL C00473 V=150.0
MOVL C00474 V=150.0
MOVL C00475 V=150.0
MOVL C00476 V=150.0
MOVL C00477 V=150.0
MOVL C00478 V=150.0
MOVL C00479 V=150.0
MOVL C00480 V=150.0
MOVL C00481 V=150.0
MOVL C00482 V=150.0
MOVL C00483 V=150.0
MOVL C00484 V=150.0
MOVL C00485 V=150.0
MOVL C00486 V=150.0
MOVL C00487 V=150.0
MOVL C00488 V=150.0
MOVL C00489 V=150.0
MOVL C00490 V=150.0
MOVL C00491 V=150.0
MOVL C00492 V=150.0
MOVL C00493 V=150.0
MOVL C00494 V=150.0
MOVL C00495 V=150.0
MOVL C00496 V=150.0
MOVL C00497 V=150.0
MOVL C00498 V=150.0
MOVL C00499 V=150.0
MOVL C00500 V=150.0
MOVL C00501 V=150.0
MOVL C00502 V=150.0
MOVL C00503 V=150.0
MOVL C00504 V=150.0
MOVL C00505 V=150.0
MOVL C00506 V=150.0
MOVL C00507 V=150.0
MOVL C00508 V=150.0
MOVL C00509 V=150.0
MOVL C00510 V=150.0
MOVL C00511 V=150.0
MOVL C00512 V=150.0
MOVL C00513 V=150.0
MOVL C00514 V=150.0
MOVL C00515 V=150.0
MOVL C00516 V=150.0
MOVL C00517 V=150.0
MOVL C00518 V=150.0
MOVL C00519 V=150.0
MOVL C00520 V=150.0
MOVL C00521 V=150.0
MOVL C00522 V=150.0
MOVL C00523 V=150.0
MOVL C00524 V=150.0
MOVL C00525 V=150.0
MOVL C00526 V=150.0
MOVL C00527 V=150.0
MOVL C00528 V=150.0
MOVL C00529 V=150.0
MOVL C00530 V=150.0
MOVL C00531 V=150.0
MOVL C00532 V=150.0
MOVL C00533 V=150.0
MOVL C00534 V=150.0
MOVL C00535 V=150.0
MOVL C00536 V=150.0
MOVL C00537 V=150.0
MOVL C00538 V=150.0
MOVL C00539 V=150.0
MOVL C00540 V=150.0
MOVL C00541 V=150.0
MOVL C00542 V=150.0
MOVL C00543 V=150.0
MOVL C00544 V=150.0
MOVL C00545 V=150.0
MOVL C00546 V=150.0
MOVL C00547 V=150.0
MOVL C00548 V=150.0
MOVL C00549 V=150.0
MOVL C00550 V=150.0
MOVL C00551 V=150.0
MOVL C00552 V=150.0
MOVL C00553 V=150.0
MOVL C00554 V=150.0
MOVL C00555 V=150.0
MOVL C00556 V=150.0
MOVL C00557 V=150.0
MOVL C00558 V=150.0
MOVL C00559 V=150.0
MOVL C00560 V=150.0
MOVL C00561 V=150.0
MOVL C00562 V=150.0
MOVL C00563 V=150.0
MOVL C00564 V=150.0
MOVL C00565 V=150.0
MOVL C00566 V=150.0
MOVL C00567 V=150.0
MOVL C00568 V=150.0
MOVL C00569 V=150.0
MOVL C00570 V=150.0
MOVL C00571 V=150.0
MOVL C00572 V=150.0
MOVL C00573 V=150.0
MOVL C00574 V=150.0
MOVL C00575 V=150.0
MOVL C00576 V=150.0
MOVL C00577 V=150.0
MOVL C00578 V=150.0
MOVL C00579 V=150.0
MOVL C00580 V=150.0
MOVL C00581 V=150.0
MOVL C00582 V=150.0
MOVL C00583 V=150.0
MOVL C00584 V=150.0
MOVL C00585 V=150.0
MOVL C00586 V=150.0
MOVL C00587 V=150.0
MOVL C00588 V=150.0
MOVL C00589 V=150.0
MOVL C00590 V=150.0
MOVL C00591 V=150.0
MOVL C00592 V=150.0
MOVL C00593 V=150.0
MOVL C00594 V=150.0
MOVL C00595 V=150.0
MOVL C00596 V=150.0
MOVL C00597 V=150.0
MOVL C00598 V=150.0
MOVL C00599 V=150.0
MOVL C00600 V=150.0
MOVL C00601 V=150.0
MOVL C00602 V=150.0
MOVL C00603 V=150.0
MOVL C00604 V=150.0
MOVL C00605 V=150.0
MOVL C00606 V=150.0
MOVL C00607 V=150.0
MOVL C00608 V=150.0
MOVL C00609 V=150.0
MOVL C00610 V=150.0
MOVL C00611 V=150.0
MOVL C00612 V=150.0
MOVL C00613 V=150.0
MOVL C00614 V=150.0
MOVL C00615 V=150.0
MOVL C00616 V=150.0
MOVL C00617 V=150.0
MOVL C00618 V=150.0
MOVL C00619 V=150.0
END
